FUNCTION_BLOCK FB_HE_SolidAttenuator EXTENDS FB_Fallible
VAR CONSTANT
    nNumHolders : INT := 5;
END_VAR
VAR
    iConvertUnits : I_ConvertUnitsLREAL;
    iSettings : I_HE_SolidAttenuatorSettings;
    iCommands : I_HE_SolidAttenuatorCommands;
    iBeamPhotonEnergy : I_QuantityLREAL;
    iBeamEnergy : I_QuantityLREAL;
    iBeamRepetitionRate : I_QuantityLREAL;
    iRequestedTransmission : I_QuantityLREAL;
    iThicknessCalculator : I_CalcThicknessFromXRayTransmission;
    iTransmissionCalculator : I_CalcXRayTransmissionFromThickness;
    iAbsorptionConstantCalculator : I_CalcXRayAbsorptionConstant;
    aiHolder : ARRAY[1..nNumHolders] OF I_HE_SolidAttenuatorHolder;

    fbCalculatedTransmission : FB_QuantityLREALPublic(Units := '1');
    fbCalculatedIncidentBeamPower : FB_QuantityLREALPublic(Units := 'W');
    fbSiliconSafeIncidentPower : FB_QuantityLREALPublic(Units := 'W');
    aiFiltersSelected : ARRAY[1..nNumHolders] OF I_HE_SolidAttenuatorFilter;

    stSettings : ST_HE_SolidAttenuatorSettings;
    nIndex : INT;
    sMaterialFormula : T_MaxString;
    fbThickness : FB_QuantityLREALPublic(Units := 'um');
    afbCalculatedTransmissionBasedOnHolderPositions : ARRAY[1..nNumHolders] OF FB_QuantityLREALPublic(Units := '1');
    fbCalculatedTransmissionBasedOnHolderPositionsTotal : FB_QuantityLREALPublic(Units := '1');

    fbAbsorptionConstant : FB_QuantityLREALPublic(Units := '1/um');
    fbSiliconThicknessRequired : FB_QuantityLREALPublic(Units := 'um');
    fbDiamondThicknessRequired : FB_QuantityLREALPublic(Units := 'um');

    eCommand : E_HE_SolidAttenuatorCommand;
END_VAR


GetSettings(Settings := stSettings);

IF NOT stSettings.bEnabled THEN
    RETURN;
END_IF

CalculateTransmissionBasedOnHolderPositions(
    CalculatedTransmission := fbCalculatedTransmission
);

CalculateIncidentBeamPower(
    BeamEnergy := iBeamEnergy,
    BeamRepetitionRate := iBeamRepetitionRate,
    BeamPowerReductionFactorAtSATTLocation := stSettings.fbBeamPowerReductionFactorAtSATTLocation,
    CalculatedIncidentBeamPower := fbCalculatedIncidentBeamPower
);

IF NOT iCommands.HasNewCommand() THEN
    RETURN;
END_IF

CASE eCommand OF
    E_HE_SolidAttenuatorCommand.CALCULATE:
        DetermineFilterSelectionForTransmission(
            RequestedTransmission := iRequestedTransmission,
            FiltersSelected := aiFiltersSelected
        );
    E_HE_SolidAttenuatorCommand.GO:
        MoveToSelectedSlots(
            HolderA1 := aiHolder[1],
            HolderA2 := aiHolder[2],
            HolderA3 := aiHolder[3],
            HolderA4 := aiHolder[4],
            HolderA5 := aiHolder[5],
            FiltersSelected := aiFiltersSelected
        );
END_CASE


METHOD CalculateDiamondThicknessForSafeSilicon
VAR_INPUT
END_VAR
END_METHOD


METHOD CalculateDiamondThicknessRequiredForTransmission
VAR_INPUT
    Transmission : I_QuantityLREAL;
    DiamondThicknessRequired : I_QuantityLREALPublic;
END_VAR
END_METHOD


METHOD CalculateIncidentBeamPower
VAR_INPUT
    BeamEnergy : I_QuantityLREAL;
    BeamRepetitionRate : I_QuantityLREAL;
    BeamPowerReductionFactorAtSATTLocation : I_QuantityLREAL;
    CalculatedIncidentBeamPower : I_QuantityLREALPublic;
END_VAR

// TODO: Unit Check

CalculatedIncidentBeamPower.Val :=
    BeamEnergy.Val *
    BeamRepetitionRate.Val *
    BeamPowerReductionFactorAtSATTLocation.Val;
END_METHOD


METHOD CalculateSiliconThicknessRequired
VAR_INPUT
    Transmission : I_QuantityLREAL;
    SiliconThicknessRequired : I_QuantityLREALPublic;
END_VAR
END_METHOD


METHOD CalculateThicknessRequiredForRequestedTransmission
VAR_INPUT
    MaterialFormula : T_MaxString;
    RequestedTransmission : I_QuantityLREAL;
    ThicknessRequired : I_QuantityLREALPublic;
END_VAR

iAbsorptionConstantCalculator.Calculate(
    MaterialFormula := MaterialFormula,
    AbsorptionConstant := fbAbsorptionConstant
);

IF iAbsorptionConstantCalculator.GetError() THEN
    SetError(Msg :=
        CONCAT('Error when attempting to calculate absorption constant: ',
        iAbsorptionConstantCalculator.GetErrorMsg()));
    RETURN;
END_IF

// TODO handle 0 absorption constant case.

ThicknessRequired.Val := LN(1.0 / RequestedTransmission.Val) / fbAbsorptionConstant.Val;
END_METHOD


METHOD CalculateTransmissionBasedOnHolderPositions
VAR_INPUT
    CalculatedTransmission : I_QuantityLREALPublic;
END_VAR

CalculatedTransmission.Val := 1.0;

FOR nIndex := 1 TO nNumHolders BY 1 DO
    aiHolder[nIndex].GetMaterialAtBeamPosition(Material := sMaterialFormula);

    aiHolder[nIndex].GetThicknessAtBeamPosition(Thickness := fbThickness);

    iTransmissionCalculator.Calculate(
        MaterialFormula := sMaterialFormula,
        Thickness := fbThickness,
        Transmission := afbCalculatedTransmissionBasedOnHolderPositions[nIndex]
    );

    CalculatedTransmission.Val :=
        fbCalculatedTransmissionBasedOnHolderPositionsTotal.Val *
        afbCalculatedTransmissionBasedOnHolderPositions[nIndex];
END_FOR
END_METHOD


METHOD PRIVATE ClearFilterSelections
END_METHOD


METHOD DetermineFilterSelectionForTransmission
VAR_INPUT
    RequestedTransmission : I_QuantityLREAL;
    FiltersSelected : ARRAY[1..nNumHolders] OF I_HE_SolidAttenuatorFilter;
END_VAR

GetSettings(Settings := stSettings);

ClearFilterSelections();

IF RequestedTransmission.Val <= 0.0 THEN
    // Return thickest arrangement.
    SelectThickestDiamondFilters(
        FiltersSelected := aiFiltersSelected
    );
    RETURN;
END_IF

CalculateSiliconThicknessRequired(
    Transmission := RequestedTransmission,
    SiliconThicknessRequired := fbSiliconThicknessRequired
);

IF fbSiliconThicknessRequired.Val < stSettings.fbDiamondOnlySiliconThicknessThreshold.Val THEN
    // If the silicon thickness required is less than the threshold, we need to only use diamond.
    // Calculate Diamond Thickness Required
    CalculateDiamondThicknessRequiredForTransmission(
        Transmission := RequestedTransmission,
        DiamondThicknessRequired := fbDiamondThicknessRequired
    );

    SelectDiamondFilters(
        ThicknessDesired := fbDiamondThicknessRequired,
        RoundingMode := stSettings.eRoundingMode,
        FiltersSelected := aiFiltersSelected,
        ThicknessSelected := fbDiamondThicknessSelected,
        TransmissionOfSelection := fbTransmissionOfSelectedDiamond
    );

    RETURN;
ELSIF fbSiliconThicknessRequired.Val >= stSettings.fbDiamondOnlySiliconThicknessThreshold.Val AND
    fbSiliconThicknessRequired.Val < stSettings.fbGermaniumNeededSiliconThicknessThreshold.Val
    // If we are above the diamond only threshold but under the germanium threshold, we use silicon only or silicon with diamond.
    // Calculate if diamond prefilter required and calculate silcon thickness required
    CalculateSafeIncidentPowerThresholdForSiliconThickness(
        PhotonEnergy := iBeamPhotonEnergy,
        SiliconThickness := fbSiliconThicknessRequired,
        SafeIncidentPower := fbSiliconSafeIncidentPower
    );

    IF fbCalculatedIncidentBeamPower.Val < fbSiliconSafeIncidentPower.Val THEN
        // We are OK with just the silicon.
        SelectSiliconFilters(
            ThicknessDesired := fbSiliconThicknessRequired,
            RoundingMode := stSettings.eRoundingMode,
            FiltersSelected := aiFiltersSelected,
            ThicknessSelected := fbSiliconThicknessSelected,
            TransmissionOfSelection := fbTransmissionOfSelectedSilicon
        );

        RETURN;
    ELSE
        // We need diamond prefilters to protect the silicon.
        // Calculate diamond filters required to protect silicon, then iterate on
        // silicon thickness to get diamond filters required to achieve transmission,
        // then check if the new silicon thickness is still protected by the diamond filters,
        // iterate until all conditions are satisfied.
        WHILE fbCalculatedIncidentBeamPower.Val > fbSiliconSafeIncidentPower.Val DO
            CalculateTransmissionRequiredForSafeFilter(
                IncidentPower := fbCalculatedIncidentBeamPower,
                SafeIncidentPower := fbSiliconSafeIncidentPower,
                RequiredTransmissionForSafeFilter := fbRequiredTransmissionForSafeSilicon
            );

            CalculateDiamondThicknessRequiredForTransmission(
                Transmission := fbRequiredTransmissionForSafeSilicon,
                DiamondThicknessRequired := fbDiamondThicknessRequired
            );

            SelectDiamondFilters(
                ThicknessDesired := fbDiamondThicknessRequired,
                RoundingMode := E_HE_SolidAttenuatorCalculationMode.CEILING,
                FiltersSelected := aiFiltersSelected,
                ThicknessSelected := fbDiamondThicknessSelected,
                TransmissionOfSelection := fbTransmissionOfSelectedDiamond
            );

            fbRequiredTransmissionForSiliconAfterDiamond.Val :=
                RequestedTransmission.Val /
                fbTransmissionOfSelectedDiamond.Val;

            CalculateSiliconThicknessRequiredForTransmission(
                Transmission := fbRequiredTransmissionForSiliconAfterDiamond,
                SiliconThicknessRequired := fbSiliconThicknessRequired
            );

            SelectSiliconFilters(
                ThicknessDesired := fbSiliconThicknessRequired,
                RoundingMode := stSettings.eRoundingMode,
                FiltersSelected := aiFiltersSelected,
                ThicknessSelected := fbSiliconThicknessSelected,
                TransmissionOfSelection := fbTransmissionOfSelectedSilicon
            );

            CalculateSafeIncidentPowerThresholdForSiliconThickness(
                PhotonEnergy := iBeamPhotonEnergy,
                SiliconThickness := fbSiliconThicknessRequired,
                SafeIncidentPower := fbSiliconSafeIncidentPower
            );
        END_WHILE
    END_IF
ELSE
    // Calculate germanium thickness required to be used with 3000um of Silicon thickness

END_IF
END_METHOD


METHOD FB_Init: BOOL
VAR_INPUT
    bInitRetains: BOOL; // TRUE: the retain variables are initialized (reset warm / reset cold)
    bInCopyCode: BOOL;  // TRUE: the instance will be copied to the copy code afterward (online change)

    ConvertUnits : I_ConvertUnitsLREAL;
    Settings : I_HE_SolidAttenuatorSettings;
    Commands : I_HE_SolidAttenuatorCommands;
    BeamPhotonEnergy : I_QuantityLREAL;
    BeamEnergy : I_QuantityLREAL;
    BeamRepetitionRate : I_QuantityLREAL;
    RequestedTransmission : I_QuantityLREAL;
    ThicknessCalculator : I_CalcThicknessFromXRayTransmission;
    TransmissionCalculator : I_CalcXRayTransmissionFromThickness;
    AbsorptionConstantCalculator : I_CalcXRayAbsorptionConstant;
    HolderA1 : I_HE_SolidAttenuatorHolder;
    HolderA2 : I_HE_SolidAttenuatorHolder;
    HolderA3 : I_HE_SolidAttenuatorHolder;
    HolderA4 : I_HE_SolidAttenuatorHolder;
    HolderA5 : I_HE_SolidAttenuatorHolder;
END_VAR

iConvertUnits := ConvertUnits;
iSettings := Settings;
iCommands := Commands;
iBeamPhotonEnergy := BeamPhotonEnergy;
iBeamEnergy := BeamEnergy;
iBeamRepetitionRate := BeamRepetitionRate;
iRequestedTransmission := RequestedTransmission;
iThicknessCalculator := ThicknessCalculator;
iTransmissionCalculator := TransmissionCalculator;
iAbsorptionConstantCalculator := AbsorptionConstantCalculator;
aiHolder[1] := HolderA1;
aiHolder[2] := HolderA2;
aiHolder[3] := HolderA3;
aiHolder[4] := HolderA4;
aiHolder[5] := HolderA5;
END_METHOD

{warning 'Add method implementation '}
METHOD GetSettings
VAR_IN_OUT
    Settings	: ST_HE_SolidAttenuatorSettings;
END_VAR
END_METHOD

METHOD IsBeamOff : BOOL
VAR_INPUT
END_VAR
END_METHOD


METHOD MoveToSelectedSlots
VAR_INPUT
    HolderA1 : I_HE_SolidAttenuatorHolder;
    HolderA2 : I_HE_SolidAttenuatorHolder;
    HolderA3 : I_HE_SolidAttenuatorHolder;
    HolderA4 : I_HE_SolidAttenuatorHolder;
    HolderA5 : I_HE_SolidAttenuatorHolder;
    aiFiltersSelected : ARRAY[1..nNumHolders] OF I_HE_SolidAttenuatorFilter;
END_VAR
END_METHOD

METHOD RequestBeamOff
VAR_INPUT
END_VAR
END_METHOD


METHOD SelectSlotsWithThickestFilters
VAR_INPUT
    HolderSlotsSelected := aiHolderSlotsSelected,
    TransmissionOfSelection := fbTransmissionOfSelected
END_VAR
END_METHOD


METHOD SelectThickestDiamondFilters
VAR_IN_OUT
    FiltersSelected : ARRAY[1..nNumHolders] OF I_HE_SolidAttenuatorFilter;
END_VAR
END_METHOD

END_FUNCTION_BLOCK

(* stored: Version 1.1.0.1
   POU FB_HE_SolidAttenuator: Id {0308bf0b-9079-42fc-a6b3-8754767b71e7}, SpecialFunc None
   Method CalculateDiamondThicknessForSafeSilicon: Id {00e08ca7-9f27-439f-bdfd-c5f1be874ee5}
   Method CalculateDiamondThicknessRequiredForTransmission: Id {ed9b5450-43f2-4302-8ff7-a671681a566e}
   Method CalculateIncidentBeamPower: Id {a2c28c84-8b19-4ceb-8725-dc51f2fd4c75}
   Method CalculateSiliconThicknessRequired: Id {ed45e70f-44b7-4a8b-8c7e-9b6580e19f18}
   Method CalculateThicknessRequiredForRequestedTransmission: Id {6690e18b-82cf-4b13-97d4-ceee8473cbc3}
   Method CalculateTransmissionBasedOnHolderPositions: Id {01f62865-349d-4382-956f-50a7d7142091}
   Method ClearFilterSelections: Id {9decf173-eeb3-4b61-b14c-dabc09381c40}
   Method DetermineFilterSelectionForTransmission: Id {e7c3860a-04b1-4dad-be3e-4cea142932dd}
   Method FB_Init: Id {6acfac08-5f66-4b17-825d-f8678fa991c3}
   Method GetSettings: Id {2f8f58b3-5f5a-49c0-828f-a8647db0ea56}
   Method IsBeamOff: Id {2e887466-2078-4dcc-90df-9f9a42ba3e4f}
   Method MoveToSelectedSlots: Id {4ae30c08-7db8-4db9-a535-c51d673bd1c9}
   Method RequestBeamOff: Id {1054a9f5-9f34-4b62-bbaf-654b23a0f45b}
   Method SelectSlotsWithThickestFilters: Id {de3a8c16-d720-451e-92cf-fb4b11929598}
   Method SelectThickestDiamondFilters: Id {f22dabb0-6900-4cbe-a015-f0065932f1ba} *)
